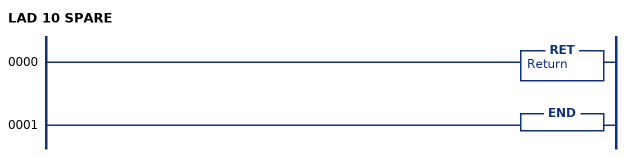
% Rung: 0 %
SOR RET EOR
% Rung: 1 %
SOR END EOR

LADDER 11 "STAGING"
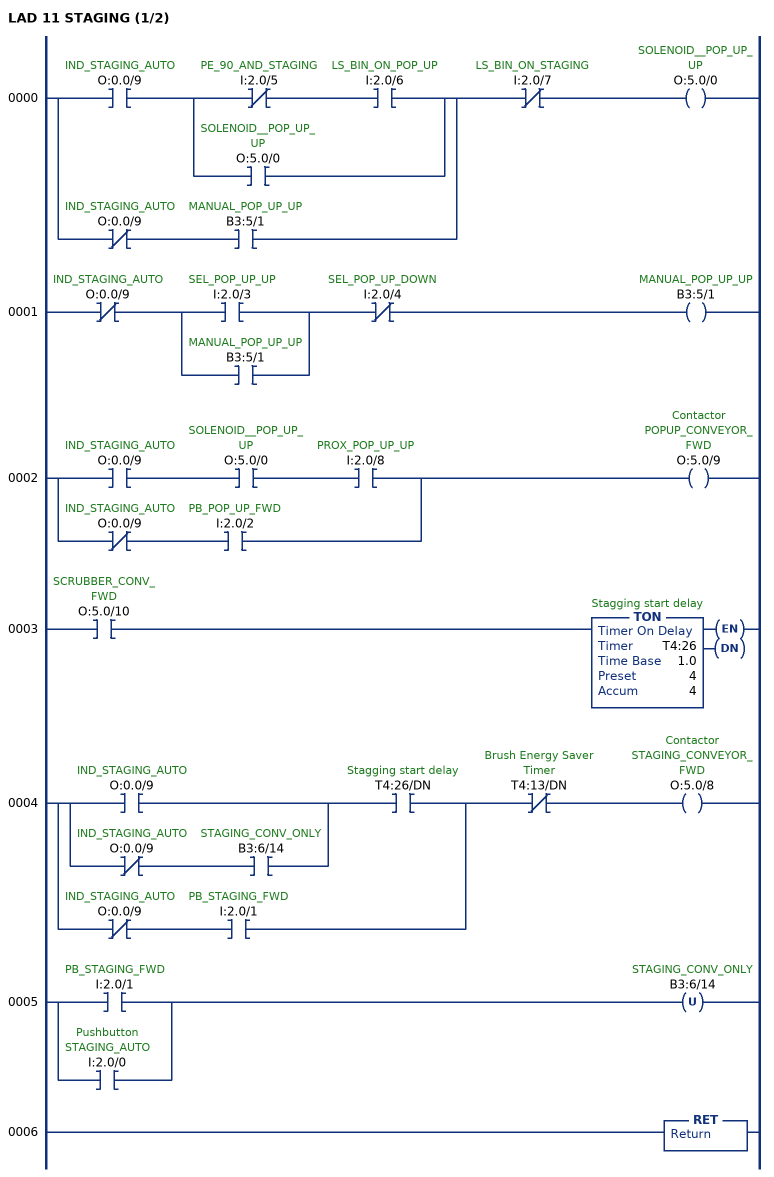
% Rung: 0 %
SOR BST XIC O:0.0/9 BST XIO I:2.0/5 XIC I:2.0/6 NXB XIC O:5.0/0 BND NXB XIO O:0.0/9 XIC B3:5/1 BND XIO I:2.0/7 OTE O:5.0/0 EOR
%   O:0.0/9  IND_STAGING_AUTO %
%   I:2.0/5  PE_90_AND_STAGING %
%   I:2.0/6  LS_BIN_ON_POP_UP %
%   O:5.0/0  SOLENOID__POP_UP_UP %
%   B3:5/1  MANUAL_POP_UP_UP %
%   I:2.0/7  LS_BIN_ON_STAGING %
% Rung: 1 %
SOR XIO O:0.0/9 BST XIC I:2.0/3 NXB XIC B3:5/1 BND XIO I:2.0/4 OTE B3:5/1 EOR
%   O:0.0/9  IND_STAGING_AUTO %
%   I:2.0/3  SEL_POP_UP_UP %
%   B3:5/1  MANUAL_POP_UP_UP %
%   I:2.0/4  SEL_POP_UP_DOWN %
% Rung: 2 %
SOR BST XIC O:0.0/9 XIC O:5.0/0 XIC I:2.0/8 NXB XIO O:0.0/9 XIC I:2.0/2 BND OTE O:5.0/9 EOR
%   O:0.0/9  IND_STAGING_AUTO %
%   O:5.0/0  SOLENOID__POP_UP_UP %
%   I:2.0/8  PROX_POP_UP_UP %
%   I:2.0/2  PB_POP_UP_FWD %
%   O:5.0/9  POPUP_CONVEYOR_FWD  "Contactor" %
% Rung: 3 %
SOR XIC O:5.0/10 TON T4:26 1.0 4 4 EOR
%   O:5.0/10  SCRUBBER_CONV_FWD %
%   T4:26  "Stagging start delay" %
% Rung: 4 %
SOR BST BST XIC O:0.0/9 NXB XIO O:0.0/9 XIC B3:6/14 BND XIC T4:26/DN NXB XIO O:0.0/9 XIC I:2.0/1 BND XIO T4:13/DN OTE O:5.0/8 EOR
%   O:0.0/9  IND_STAGING_AUTO %
%   B3:6/14  STAGING_CONV_ONLY %
%   T4:26  "Stagging start delay" %
%   I:2.0/1  PB_STAGING_FWD %
%   T4:13  "Brush Energy Saver Timer" %
%   O:5.0/8  STAGING_CONVEYOR_FWD  "Contactor" %
% Rung: 5 %
SOR BST XIC I:2.0/1 NXB XIC I:2.0/0 BND OTU B3:6/14 EOR
%   I:2.0/1  PB_STAGING_FWD %
%   I:2.0/0  STAGING_AUTO  "Pushbutton" %
%   B3:6/14  STAGING_CONV_ONLY %
% Rung: 6 %
SOR RET EOR

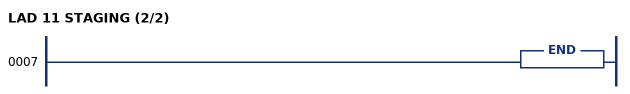
% Rung: 7 %
SOR END EOR

LADDER 12 "DESTACK LS"
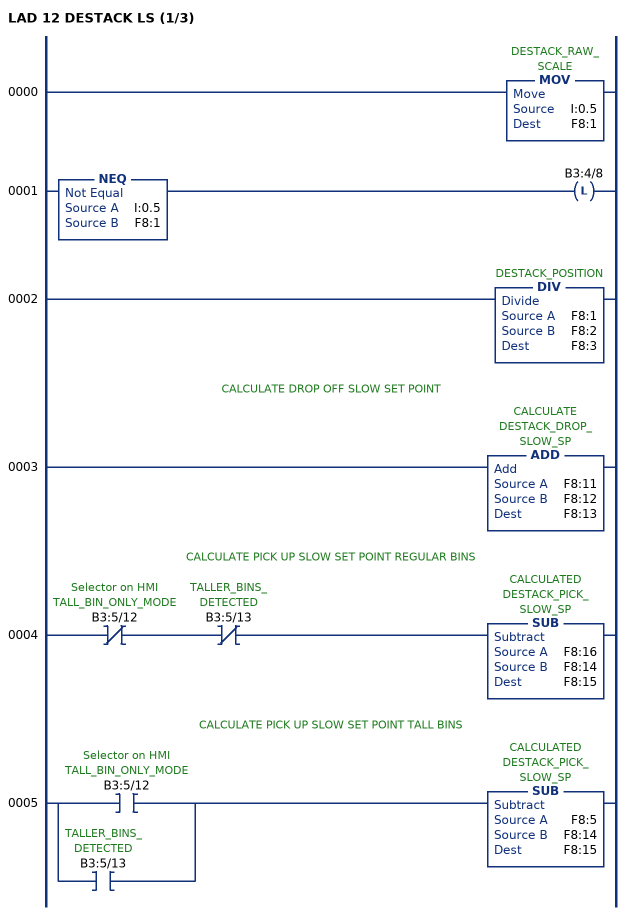
% Rung: 0 %
SOR MOV I:0.5 F8:1 EOR
%   F8:1  DESTACK_RAW_SCALE %
% Rung: 1 %
SOR NEQ I:0.5 F8:1 OTL B3:4/8 EOR
%   F8:1  DESTACK_RAW_SCALE %
%   OTL B3:4/8  "ANALOG FAULT" %
% Rung: 2 %
SOR DIV F8:1 F8:2 F8:3 EOR
%   F8:1  DESTACK_RAW_SCALE %
%   F8:2  DESTACK_SCALLER %
%   F8:3  DESTACK_POSITION %
% Rung: 3 %
% CALCULATE DROP OFF SLOW SET POINT %
SOR ADD F8:11 F8:12 F8:13 EOR
%   F8:11  DESTACK_DROP_OFF_SP  "ACTUAL" %
%   F8:12  DESTACK_DROP_SLOW  "OFFSET" %
%   F8:13  DESTACK_DROP_SLOW_SP  "CALCULATE" %
% Rung: 4 %
% CALCULATE PICK UP SLOW SET POINT REGULAR BINS %
SOR XIO B3:5/12 XIO B3:5/13 SUB F8:16 F8:14 F8:15 EOR
%   B3:5/12  TALL_BIN_ONLY_MODE  "Selector on HMI" %
%   B3:5/13  TALLER_BINS_DETECTED %
%   F8:16  PICK_UP_SP  "ACTUAL" %
%   F8:14  DESTACK_PU_SLOW  "OFFSET" %
%   F8:15  DESTACK_PICK_SLOW_SP  "CALCULATED" %
% Rung: 5 %
% CALCULATE PICK UP SLOW SET POINT TALL BINS %
SOR BST XIC B3:5/12 NXB XIC B3:5/13 BND SUB F8:5 F8:14 F8:15 EOR
%   B3:5/12  TALL_BIN_ONLY_MODE  "Selector on HMI" %
%   B3:5/13  TALLER_BINS_DETECTED %
%   F8:5  TALL_BIN_PU_POSITION %
%   F8:14  DESTACK_PU_SLOW  "OFFSET" %
%   F8:15  DESTACK_PICK_SLOW_SP  "CALCULATED" %

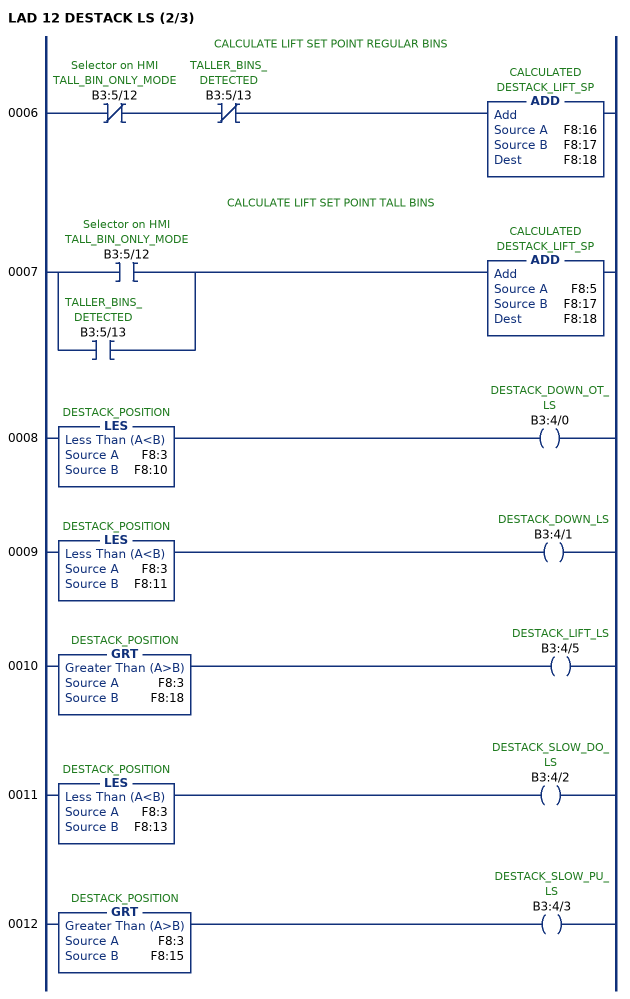
% Rung: 6 %
% CALCULATE LIFT SET POINT REGULAR BINS %
SOR XIO B3:5/12 XIO B3:5/13 ADD F8:16 F8:17 F8:18 EOR
%   B3:5/12  TALL_BIN_ONLY_MODE  "Selector on HMI" %
%   B3:5/13  TALLER_BINS_DETECTED %
%   F8:16  PICK_UP_SP  "ACTUAL" %
%   F8:17  DESTACK_LIFT  "OFFSET" %
%   F8:18  DESTACK_LIFT_SP  "CALCULATED" %
% Rung: 7 %
% CALCULATE LIFT SET POINT TALL BINS %
SOR BST XIC B3:5/12 NXB XIC B3:5/13 BND ADD F8:5 F8:17 F8:18 EOR
%   B3:5/12  TALL_BIN_ONLY_MODE  "Selector on HMI" %
%   B3:5/13  TALLER_BINS_DETECTED %
%   F8:5  TALL_BIN_PU_POSITION %
%   F8:17  DESTACK_LIFT  "OFFSET" %
%   F8:18  DESTACK_LIFT_SP  "CALCULATED" %
% Rung: 8 %
SOR LES F8:3 F8:10 OTE B3:4/0 EOR
%   F8:3  DESTACK_POSITION %
%   F8:10  DESTACK_LOWER_OT_SP  "ACTUAL" %
%   B3:4/0  DESTACK_DOWN_OT_LS %
% Rung: 9 %
SOR LES F8:3 F8:11 OTE B3:4/1 EOR
%   F8:3  DESTACK_POSITION %
%   F8:11  DESTACK_DROP_OFF_SP  "ACTUAL" %
%   B3:4/1  DESTACK_DOWN_LS %
% Rung: 10 %
SOR GRT F8:3 F8:18 OTE B3:4/5 EOR
%   F8:3  DESTACK_POSITION %
%   F8:18  DESTACK_LIFT_SP  "CALCULATED" %
%   B3:4/5  DESTACK_LIFT_LS %
% Rung: 11 %
SOR LES F8:3 F8:13 OTE B3:4/2 EOR
%   F8:3  DESTACK_POSITION %
%   F8:13  DESTACK_DROP_SLOW_SP  "CALCULATE" %
%   B3:4/2  DESTACK_SLOW_DO_LS %
% Rung: 12 %
SOR GRT F8:3 F8:15 OTE B3:4/3 EOR
%   F8:3  DESTACK_POSITION %
%   F8:15  DESTACK_PICK_SLOW_SP  "CALCULATED" %
%   B3:4/3  DESTACK_SLOW_PU_LS %

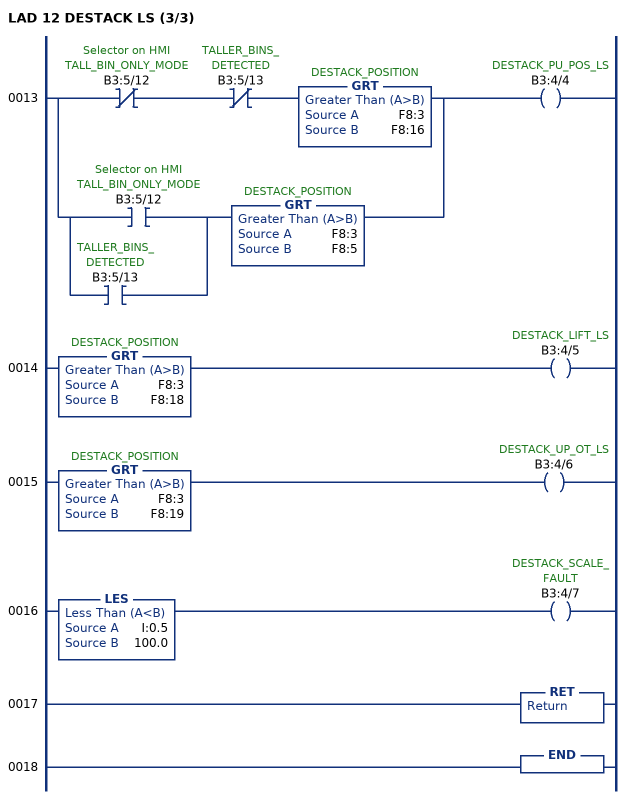
% Rung: 13 %
SOR BST XIO B3:5/12 XIO B3:5/13 GRT F8:3 F8:16 NXB BST XIC B3:5/12 NXB XIC B3:5/13 BND GRT F8:3 F8:5 BND OTE B3:4/4 EOR
%   B3:5/12  TALL_BIN_ONLY_MODE  "Selector on HMI" %
%   B3:5/13  TALLER_BINS_DETECTED %
%   F8:3  DESTACK_POSITION %
%   F8:16  PICK_UP_SP  "ACTUAL" %
%   F8:5  TALL_BIN_PU_POSITION %
%   B3:4/4  DESTACK_PU_POS_LS %
% Rung: 14 %
SOR GRT F8:3 F8:18 OTE B3:4/5 EOR
%   F8:3  DESTACK_POSITION %
%   F8:18  DESTACK_LIFT_SP  "CALCULATED" %
%   B3:4/5  DESTACK_LIFT_LS %
% Rung: 15 %
SOR GRT F8:3 F8:19 OTE B3:4/6 EOR
%   F8:3  DESTACK_POSITION %
%   F8:19  DESTACK_UPPER_OT_SP  "ACTUAL" %
%   B3:4/6  DESTACK_UP_OT_LS %
% Rung: 16 %
SOR LES I:0.5 100.0 OTE B3:4/7 EOR
%   B3:4/7  DESTACK_SCALE_FAULT %
% Rung: 17 %
SOR RET EOR
% Rung: 18 %
SOR END EOR

LADDER 13 "DESTACK"
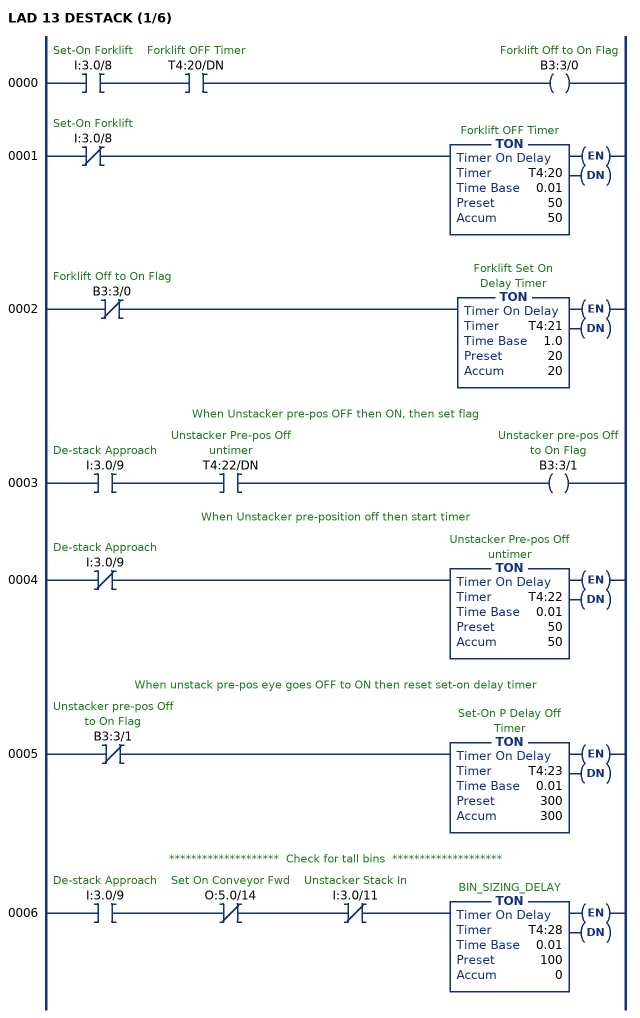
% Rung: 0 %
SOR XIC I:3.0/8 XIC T4:20/DN OTE B3:3/0 EOR
%   I:3.0/8  "Set-On Forklift" %
%   T4:20  "Forklift OFF Timer" %
%   B3:3/0  "Forklift Off to On Flag" %
% Rung: 1 %
SOR XIO I:3.0/8 TON T4:20 0.01 50 50 EOR
%   I:3.0/8  "Set-On Forklift" %
%   T4:20  "Forklift OFF Timer" %
% Rung: 2 %
SOR XIO B3:3/0 TON T4:21 1.0 20 20 EOR
%   B3:3/0  "Forklift Off to On Flag" %
%   T4:21  "Forklift Set On Delay Timer" %
% Rung: 3 %
% When Unstacker pre-pos OFF then ON, then set flag %
SOR XIC I:3.0/9 XIC T4:22/DN OTE B3:3/1 EOR
%   I:3.0/9  "De-stack Approach" %
%   T4:22  "Unstacker Pre-pos Off untimer" %
%   B3:3/1  "Unstacker pre-pos Off to On Flag" %
% Rung: 4 %
% When Unstacker pre-position off then start timer %
SOR XIO I:3.0/9 TON T4:22 0.01 50 50 EOR
%   I:3.0/9  "De-stack Approach" %
%   T4:22  "Unstacker Pre-pos Off untimer" %
% Rung: 5 %
% When unstack pre-pos eye goes OFF to ON then reset set-on delay timer %
SOR XIO B3:3/1 TON T4:23 0.01 300 300 EOR
%   B3:3/1  "Unstacker pre-pos Off to On Flag" %
%   T4:23  "Set-On P Delay Off Timer" %
% Rung: 6 %
% ********************  Check for tall bins  ******************** %
SOR XIC I:3.0/9 XIO O:5.0/14 XIO I:3.0/11 TON T4:28 0.01 100 0 EOR
%   I:3.0/9  "De-stack Approach" %
%   O:5.0/14  "Set On Conveyor Fwd" %
%   I:3.0/11  "Unstacker Stack In" %
%   T4:28  BIN_SIZING_DELAY %

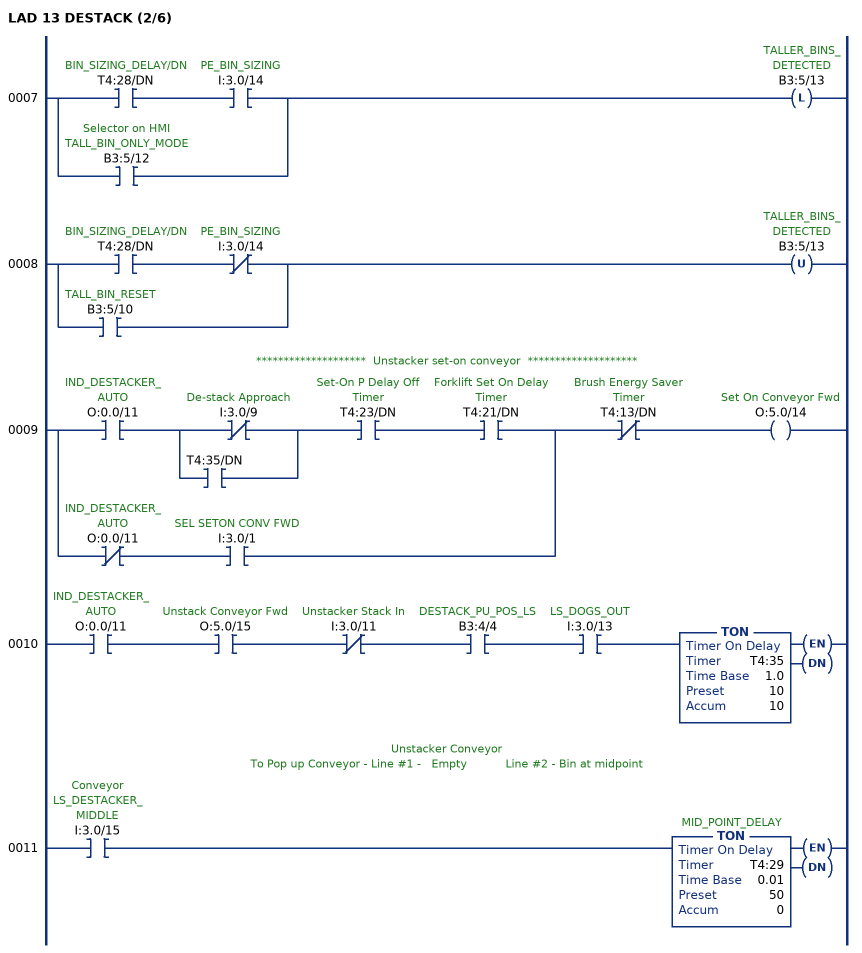
% Rung: 7 %
SOR BST XIC T4:28/DN XIC I:3.0/14 NXB XIC B3:5/12 BND OTL B3:5/13 EOR
%   T4:28  BIN_SIZING_DELAY %
%   I:3.0/14  PE_BIN_SIZING %
%   B3:5/12  TALL_BIN_ONLY_MODE  "Selector on HMI" %
%   B3:5/13  TALLER_BINS_DETECTED %
% Rung: 8 %
SOR BST XIC T4:28/DN XIO I:3.0/14 NXB XIC B3:5/10 BND OTU B3:5/13 EOR
%   T4:28  BIN_SIZING_DELAY %
%   I:3.0/14  PE_BIN_SIZING %
%   B3:5/10  TALL_BIN_RESET %
%   B3:5/13  TALLER_BINS_DETECTED %
% Rung: 9 %
% ********************  Unstacker set-on conveyor  ******************** %
SOR BST XIC O:0.0/11 BST XIO I:3.0/9 NXB XIC T4:35/DN BND XIC T4:23/DN XIC T4:21/DN NXB XIO O:0.0/11 XIC I:3.0/1 BND XIO T4:13/DN OTE O:5.0/14 EOR
%   O:0.0/11  IND_DESTACKER_AUTO %
%   I:3.0/9  "De-stack Approach" %
%   T4:23  "Set-On P Delay Off Timer" %
%   T4:21  "Forklift Set On Delay Timer" %
%   I:3.0/1  "SEL SETON CONV FWD" %
%   T4:13  "Brush Energy Saver Timer" %
%   O:5.0/14  "Set On Conveyor Fwd" %
% Rung: 10 %
SOR XIC O:0.0/11 XIC O:5.0/15 XIO I:3.0/11 XIC B3:4/4 XIC I:3.0/13 TON T4:35 1.0 10 10 EOR
%   O:0.0/11  IND_DESTACKER_AUTO %
%   O:5.0/15  "Unstack Conveyor Fwd" %
%   I:3.0/11  "Unstacker Stack In" %
%   B3:4/4  DESTACK_PU_POS_LS %
%   I:3.0/13  LS_DOGS_OUT %
% Rung: 11 %
% Unstacker Conveyor
% To Pop up Conveyor - Line #1 -   Empty           Line #2 - Bin at midpoint %
SOR XIC I:3.0/15 TON T4:29 0.01 50 0 EOR
%   I:3.0/15  LS_DESTACKER_MIDDLE  "Conveyor" %
%   T4:29  MID_POINT_DELAY %

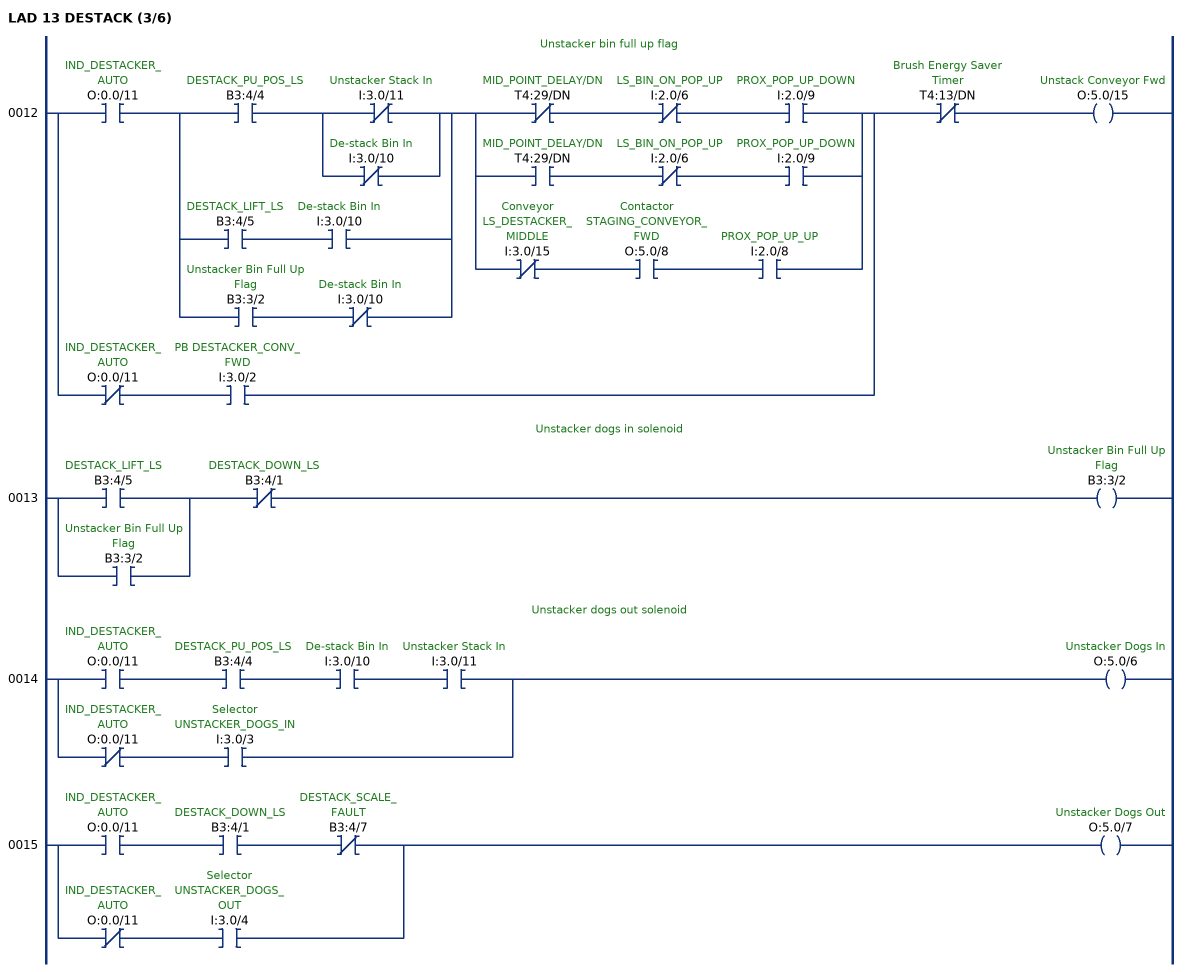
% Rung: 12 %
% Unstacker bin full up flag %
SOR BST XIC O:0.0/11 BST XIC B3:4/4 BST XIO I:3.0/11 NXB XIO I:3.0/10 BND NXB XIC B3:4/5 XIC I:3.0/10 NXB XIC B3:3/2 XIO I:3.0/10 BND BST XIO T4:29/DN XIO I:2.0/6 XIC I:2.0/9 NXB BST XIC T4:29/DN XIO I:2.0/6 XIC I:2.0/9 NXB XIO I:3.0/15 XIC O:5.0/8 XIC I:2.0/8 BND BND NXB XIO O:0.0/11 XIC I:3.0/2 BND XIO T4:13/DN OTE O:5.0/15 EOR
%   O:0.0/11  IND_DESTACKER_AUTO %
%   B3:4/4  DESTACK_PU_POS_LS %
%   I:3.0/11  "Unstacker Stack In" %
%   I:3.0/10  "De-stack Bin In" %
%   B3:4/5  DESTACK_LIFT_LS %
%   B3:3/2  "Unstacker Bin Full Up Flag" %
%   T4:29  MID_POINT_DELAY %
%   I:2.0/6  LS_BIN_ON_POP_UP %
%   I:2.0/9  PROX_POP_UP_DOWN %
%   I:3.0/15  LS_DESTACKER_MIDDLE  "Conveyor" %
%   O:5.0/8  STAGING_CONVEYOR_FWD  "Contactor" %
%   I:2.0/8  PROX_POP_UP_UP %
%   I:3.0/2  DESTACKER_CONV_FWD  "PB" %
%   T4:13  "Brush Energy Saver Timer" %
%   O:5.0/15  "Unstack Conveyor Fwd" %
% Rung: 13 %
% Unstacker dogs in solenoid %
SOR BST XIC B3:4/5 NXB XIC B3:3/2 BND XIO B3:4/1 OTE B3:3/2 EOR
%   B3:4/5  DESTACK_LIFT_LS %
%   B3:3/2  "Unstacker Bin Full Up Flag" %
%   B3:4/1  DESTACK_DOWN_LS %
% Rung: 14 %
% Unstacker dogs out solenoid %
SOR BST XIC O:0.0/11 XIC B3:4/4 XIC I:3.0/10 XIC I:3.0/11 NXB XIO O:0.0/11 XIC I:3.0/3 BND OTE O:5.0/6 EOR
%   O:0.0/11  IND_DESTACKER_AUTO %
%   B3:4/4  DESTACK_PU_POS_LS %
%   I:3.0/10  "De-stack Bin In" %
%   I:3.0/11  "Unstacker Stack In" %
%   I:3.0/3  UNSTACKER_DOGS_IN  "Selector" %
%   O:5.0/6  "Unstacker Dogs In" %
% Rung: 15 %
SOR BST XIC O:0.0/11 XIC B3:4/1 XIO B3:4/7 NXB XIO O:0.0/11 XIC I:3.0/4 BND OTE O:5.0/7 EOR
%   O:0.0/11  IND_DESTACKER_AUTO %
%   B3:4/1  DESTACK_DOWN_LS %
%   B3:4/7  DESTACK_SCALE_FAULT %
%   I:3.0/4  UNSTACKER_DOGS_OUT  "Selector" %
%   O:5.0/7  "Unstacker Dogs Out" %

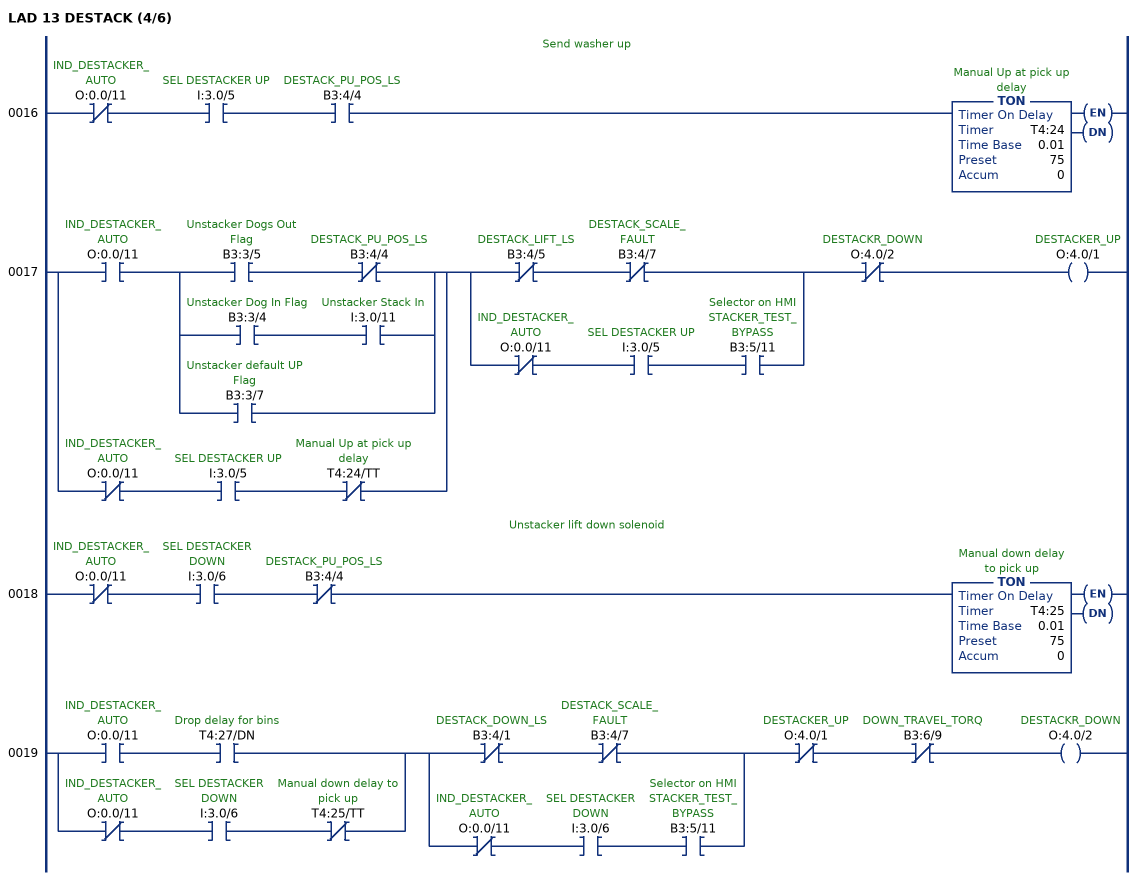
% Rung: 16 %
% Send washer up %
SOR XIO O:0.0/11 XIC I:3.0/5 XIC B3:4/4 TON T4:24 0.01 75 0 EOR
%   O:0.0/11  IND_DESTACKER_AUTO %
%   I:3.0/5  "SEL DESTACKER UP" %
%   B3:4/4  DESTACK_PU_POS_LS %
%   T4:24  "Manual Up at pick up delay" %
% Rung: 17 %
SOR BST XIC O:0.0/11 BST XIC B3:3/5 XIO B3:4/4 NXB XIC B3:3/4 XIC I:3.0/11 NXB XIC B3:3/7 BND NXB XIO O:0.0/11 XIC I:3.0/5 XIO T4:24/TT BND BST XIO B3:4/5 XIO B3:4/7 NXB XIO O:0.0/11 XIC I:3.0/5 XIC B3:5/11 BND XIO O:4.0/2 OTE O:4.0/1 EOR
%   O:0.0/11  IND_DESTACKER_AUTO %
%   B3:3/5  "Unstacker Dogs Out Flag" %
%   B3:4/4  DESTACK_PU_POS_LS %
%   B3:3/4  "Unstacker Dog In Flag" %
%   I:3.0/11  "Unstacker Stack In" %
%   B3:3/7  "Unstacker default UP Flag" %
%   I:3.0/5  "SEL DESTACKER UP" %
%   T4:24  "Manual Up at pick up delay" %
%   B3:4/5  DESTACK_LIFT_LS %
%   B3:4/7  DESTACK_SCALE_FAULT %
%   B3:5/11  STACKER_TEST_BYPASS  "Selector on HMI" %
%   O:4.0/2  DESTACKR_DOWN %
%   O:4.0/1  DESTACKER_UP %
% Rung: 18 %
% Unstacker lift down solenoid %
SOR XIO O:0.0/11 XIC I:3.0/6 XIO B3:4/4 TON T4:25 0.01 75 0 EOR
%   O:0.0/11  IND_DESTACKER_AUTO %
%   I:3.0/6  "SEL DESTACKER DOWN" %
%   B3:4/4  DESTACK_PU_POS_LS %
%   T4:25  "Manual down delay to pick up" %
% Rung: 19 %
SOR BST XIC O:0.0/11 XIC T4:27/DN NXB XIO O:0.0/11 XIC I:3.0/6 XIO T4:25/TT BND BST XIO B3:4/1 XIO B3:4/7 NXB XIO O:0.0/11 XIC I:3.0/6 XIC B3:5/11 BND XIO O:4.0/1 XIO B3:6/9 OTE O:4.0/2 EOR
%   O:0.0/11  IND_DESTACKER_AUTO %
%   T4:27  "Drop delay for bins" %
%   I:3.0/6  "SEL DESTACKER DOWN" %
%   T4:25  "Manual down delay to pick up" %
%   B3:4/1  DESTACK_DOWN_LS %
%   B3:4/7  DESTACK_SCALE_FAULT %
%   B3:5/11  STACKER_TEST_BYPASS  "Selector on HMI" %
%   O:4.0/1  DESTACKER_UP %
%   B3:6/9  DOWN_TRAVEL_TORQ %
%   O:4.0/2  DESTACKR_DOWN %

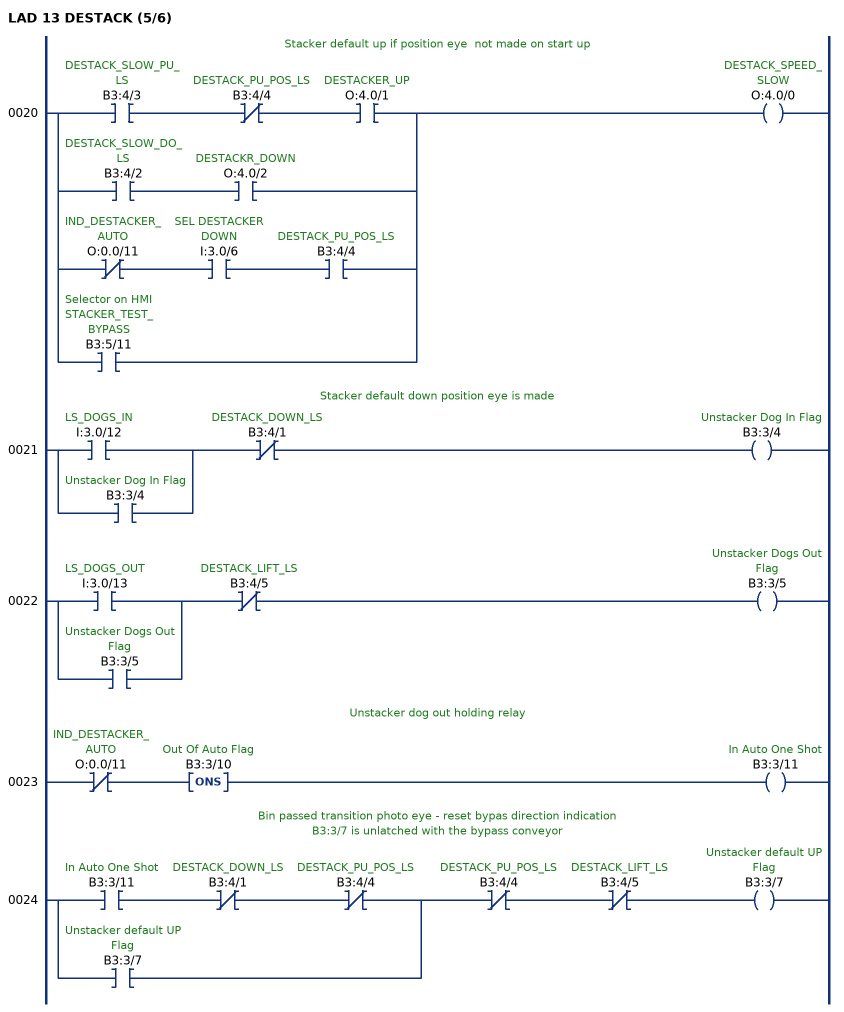
% Rung: 20 %
% Stacker default up if position eye  not made on start up %
SOR BST XIC B3:4/3 XIO B3:4/4 XIC O:4.0/1 NXB BST XIC B3:4/2 XIC O:4.0/2 NXB BST XIO O:0.0/11 XIC I:3.0/6 XIC B3:4/4 NXB XIC B3:5/11 BND BND BND OTE O:4.0/0 EOR
%   B3:4/3  DESTACK_SLOW_PU_LS %
%   B3:4/4  DESTACK_PU_POS_LS %
%   O:4.0/1  DESTACKER_UP %
%   B3:4/2  DESTACK_SLOW_DO_LS %
%   O:4.0/2  DESTACKR_DOWN %
%   O:0.0/11  IND_DESTACKER_AUTO %
%   I:3.0/6  "SEL DESTACKER DOWN" %
%   B3:5/11  STACKER_TEST_BYPASS  "Selector on HMI" %
%   O:4.0/0  DESTACK_SPEED_SLOW %
% Rung: 21 %
% Stacker default down position eye is made %
SOR BST XIC I:3.0/12 NXB XIC B3:3/4 BND XIO B3:4/1 OTE B3:3/4 EOR
%   I:3.0/12  LS_DOGS_IN %
%   B3:3/4  "Unstacker Dog In Flag" %
%   B3:4/1  DESTACK_DOWN_LS %
% Rung: 22 %
SOR BST XIC I:3.0/13 NXB XIC B3:3/5 BND XIO B3:4/5 OTE B3:3/5 EOR
%   I:3.0/13  LS_DOGS_OUT %
%   B3:3/5  "Unstacker Dogs Out Flag" %
%   B3:4/5  DESTACK_LIFT_LS %
% Rung: 23 %
% Unstacker dog out holding relay %
SOR XIO O:0.0/11 ONS B3:3/10 OTE B3:3/11 EOR
%   O:0.0/11  IND_DESTACKER_AUTO %
%   B3:3/10  "Out Of Auto Flag" %
%   B3:3/11  "In Auto One Shot" %
% Rung: 24 %
% Bin passed transition photo eye - reset bypas direction indication
% B3:3/7 is unlatched with the bypass conveyor %
SOR BST XIC B3:3/11 XIO B3:4/1 XIO B3:4/4 NXB XIC B3:3/7 BND XIO B3:4/4 XIO B3:4/5 OTE B3:3/7 EOR
%   B3:3/11  "In Auto One Shot" %
%   B3:4/1  DESTACK_DOWN_LS %
%   B3:4/4  DESTACK_PU_POS_LS %
%   B3:3/7  "Unstacker default UP Flag" %
%   B3:4/5  DESTACK_LIFT_LS %

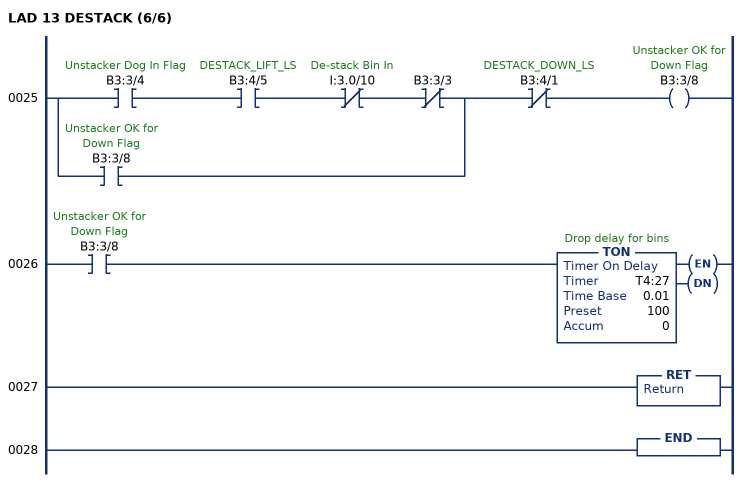
% Rung: 25 %
SOR BST XIC B3:3/4 XIC B3:4/5 XIO I:3.0/10 XIO B3:3/3 NXB XIC B3:3/8 BND XIO B3:4/1 OTE B3:3/8 EOR
%   B3:3/4  "Unstacker Dog In Flag" %
%   B3:4/5  DESTACK_LIFT_LS %
%   I:3.0/10  "De-stack Bin In" %
%   B3:3/8  "Unstacker OK for Down Flag" %
%   B3:4/1  DESTACK_DOWN_LS %
% Rung: 26 %
SOR XIC B3:3/8 TON T4:27 0.01 100 0 EOR
%   B3:3/8  "Unstacker OK for Down Flag" %
%   T4:27  "Drop delay for bins" %
% Rung: 27 %
SOR RET EOR
% Rung: 28 %
SOR END EOR

OTHER DOCUMENTED ADDRESSES
  B3:0/9  SANITIZE_LTCH  "Triggered by reset limit sw."
  B3:0/10  SANITIZE_BIT  "Allow crdl ltch2 to unlatch only once until sanitize cycle is over"
  B3:0/11  CRDL_EN  "mcr on and no encoder fault"
  B3:0/15  CRDL_HAND_SS
  B3:1/1  RINSE_SELECT  "Turn ON Rinse"
  B3:2/13  SHOW_INPUTS_OUTPUTS  "HMI"
  B3:5/0  90_AND_STAGING_BUSY
  B3:6/13  UNSTACKR_CONV_ONLY
  C5:0/CU  EVENT_COUNTER
  F8:4  TALL_BIN_OFF_SET
  I:0.4/0  DESTACK_LINER
  I:0.5/0  STACKER_LINEAR
  L10:1/1  FAULT_MESSAGES
  N7:1/0  "Fault-Infeed Blocked"
  N7:1/1  "Fault-Outfeed Blocked"
  N7:1/2  "Fault-Cradle Overtravel Up"
  N7:1/3  "Fault-Cradle Overtravel down"
  N7:1/4  "Fault-Torque Cradle Inverter"
  N7:1/5  "Main Tank Low"
  N7:1/6  "Encoder Fault"
  N7:1/7  "Fill Main Tank"
  N7:7  LOWER_WASH_TURN_OFF
  N9:0  K1
  O:0.0/7  NOT_USED
  O:2.0/1  RINSE_SOLENOID  "Rinse after wash"
  O:4.0/4  "WAS SCRUBBER CONVEYOR"
  O:5.0/3  RINSE_OPTION
  T4:0/EN  CRDL_DWN_T  "Allows cradle to set down completely before conv starts"
  T4:1  CRDL_FLT_T1
  T4:2  CRDL_FLT_T2
  T4:6  SANITIZE_T
  T4:7  CRDL_DWN_T2  "Inhibits cradle up for 5 sec. after cradle sets down"
  T4:10  CRADLE_TIMER  "Cradle travel watch dog timer"
  T4:37  GRAVITY_CONV_FULL

COMMENTS NOT ATTACHED TO A CURRENT RUNG
  N7:1/0: As long as the bit is set, the message will be displayed.  Bit #1 is Message #1.  Bit #3 is message #4.  Binary to decimal.
  T4:6.PRE: As long as the bit is set, the message will be displayed.  Bit #1 is Message #1.  Bit #3 is message #4.  Binary to decimal.
  T4:7: Timer not used
  N7:26: CALCULATE SLOW PICK UP SP
  N7:23: CALCULATE LIFT SET POINT
  N7:28: CALCULATE LIFT SET POINT
  T4:25: Looks ahead to see if the feed out conveyor is full.
  T4:24.PRE: *****************************************  HMI TABLE ROTATION ANIMATION  ******************************************************
  B3:3/9: Bin reached transition photo eye
  O:6.0/3: *******************************************************  TABLE CONVEYOR *********************************************************************
  T4:37: TURN CONVEYOR OFF WHEN FULL

REVISION NOTES
  0: Added barrier and overtravel tatches
  1: Added indepentent barrier and overtravel catches
  2: Changed ffrom Panel #8.  Added B3:0/1 to prevent B3:0/5 from latching up while cradle is not down
  3: Added more troubleshooting help - step sequences
  4: Costa Rica Panel #19 with individual upper and lower wash solenoids
  5: Changed to 1400 with additional input and output cards
  6: Aux relay
  7: aux relay

DATA TABLE (non-zero values as saved)
DATA B3
% B3:0 % 0X0D1A 0X4803 0X2838 0X0020 0X0018 0X2080 0X0008
DATA T4
% .PRE .ACC %
% T4:0 % 50 50
% T4:1 % 1 0
% T4:2 % 1 0
% T4:3 % 45 0
% T4:4 % 10 0
% T4:5 % 15 0
% T4:6 % 658 0
% T4:7 % 375 500
% T4:8 % 15 0
% T4:9 % 2 2
% T4:10 % 500 0
% T4:11 % 75 0
% T4:12 % 150 0
% T4:13 % 90 63
% T4:14 % 90 63
% T4:15 % 500 0
% T4:16 % 500 0
% T4:17 % 100 0
% T4:18 % 100 0
% T4:19 % 240 0
% T4:20 % 50 50
% T4:21 % 20 20
% T4:22 % 50 50
% T4:23 % 300 300
% T4:24 % 75 0
% T4:25 % 75 0
% T4:26 % 4 4
% T4:27 % 100 0
% T4:28 % 100 0
% T4:29 % 50 0
% T4:30 % 175 175
% T4:31 % 175 175
% T4:32 % 10 0
% T4:33 % 30 0
% T4:34 % 60 60
% T4:35 % 10 10
% T4:36 % 100 0
% T4:37 % 6 0
DATA N7
% N7:0 % 84 0 8 65 120 22 24 0 0 0
% N7:10 % 7 7 15 15 0 0 0 0 0 0
DATA F8
% F8:0 % 678 3583 104 34.45192 34.5
% F8:5 % 34 0 0 0 0
% F8:10 % 2 4 6 10 6
% F8:15 % 28 31.75 2.75 36.75 38.5
